INTERFACE I_BacklashCompensation EXTENDS I_Output

PROPERTY ActCompensation : LREAL
GET
END_GET
END_PROPERTY

(*
    Handle positive/negative backlash compensation
    User needs to set the direction of backlash from the sign of the compensation value
    Backlash compensation is disabled during referencing (homing).
    When direction is positive/negative, further movement in the negative/positive direction not compensated
    further movement in the negative/positive direction will be compensated
*)
METHOD BacklashCompensation
VAR_INPUT
    Activate     : BOOL;
    Compensation	: LREAL;
    RampVelocity	: LREAL;
    DisableMode	: E_DISABLEMODE := E_DISABLEMODE.DisableModeHold;
END_VAR
END_METHOD

(*synced Fbs need just to activate the compensation with a given ramp speed
  other parameters are provided via EPICS (declared in this FB) or via the more extended BackalshCompensation method (simulation) *)
METHOD BacklashCompensationActive
VAR_INPUT
    Active     : BOOL;
    RampVelocity : LREAL;
END_VAR
END_METHOD

PROPERTY UserEnable : BOOL
SET
END_SET
END_PROPERTY

END_INTERFACE

(* stored: Version 1.1.0.1
   Itf I_BacklashCompensation: Id {c0dc76c5-ea53-4a27-aade-dbf12ab6b44d}
   Property ActCompensation: Id {ff081112-3182-493d-846e-c2192c5f77d6}
   Get Get: Id {5dbd065d-c6db-421a-8993-7aa4f3a00024}
   Method BacklashCompensation: Id {8dc8359f-12ee-498a-aa0e-4230cfa1b09f}
   Method BacklashCompensationActive: Id {bf2a0313-baf0-4f23-9d25-649e80700102}
   Property UserEnable: Id {0e887761-1e47-4bcc-b90c-ad725d2076e6}
   Set Set: Id {87cc7722-3cc9-4268-9f17-c9fd9cad6c1f} *)
